// TwinCAT 3 PLC project PLC
// ProgramVersion: 3.1.4024.0
// libraries:
//   SPT Base Types, * (Beckhoff Automation LLC)
//   SPT Components, * (Beckhoff Automation LLC)
//   SPT Diagnostic, * (Beckhoff Automation LLC)
//   SPT EtherCat, * (Beckhoff Automation LLC)
//   SPT Event Logger, * (Beckhoff Automation LLC)
//   SPT Kinematics, * (Beckhoff Automation LLC)
//   SPT Motion Control, * (Beckhoff Automation LLC)
//   SPT NCI, * (Beckhoff Automation LLC)
//   SPT Utilities, * (Beckhoff Automation LLC)
//   SPT Vision, * (Beckhoff Automation LLC)
//   SPT XTS, * (Beckhoff Automation LLC)
//   Tc2_Standard, * (Beckhoff Automation GmbH)
//   Tc2_System, * (Beckhoff Automation GmbH)
//   Tc3_EventLogger, * (Beckhoff Automation GmbH)
//   Tc3_Module, * (Beckhoff Automation GmbH)
//   Tc3_PackML_V2, * (Beckhoff Automation GmbH)
// project tree:
//   / GlobalTextList.TcGTLO (not stored), PlcTask.TcTTO (not stored), Visualization Manager.TcVMO (not stored)
//   Machine/01_MachineModule/ Machine.TcPOU
//   Machine/02_EquipmentModules/ InfeedModule.TcPOU, OutfeedModule.TcPOU, ProcessModule.TcPOU
//   Machine/03_Components/ SampleComponent.TcPOU
//   POUs/ MAIN.TcPOU
//   VISUs/ Visualization.TcVIS
// real-time tasks:
//   TASK PlcTask: cycle T#10ms, priority 20, ADS port 350

// ---- Machine/01_MachineModule/Machine.TcPOU
FUNCTION_BLOCK Machine EXTENDS FB_PackML_BaseModule
VAR
	//EMs
	Infeed	: InfeedModule	:= (Name := 'Infeed');
	Process : ProcessModule := (Name := 'Process');
	Outfeed : OutfeedModule := (Name := 'Outfeed');

	//
	_StopRequestFromEM : BOOL;
END_VAR

//! @summary This method serves as the entry point for all underlying FB logic

//! @description This method should be called cyclically by descendant function blocks by invoking <c>SUPER^.CyclicLogic()</c>.  Alternatively, the contents of this method could be reimplemented entirely in which case a call to this method would not be necessary.
METHOD PUBLIC CyclicLogic
VAR
	i : UDINT;
END_VAR
IF NOT _InitComplete THEN
	_InitComplete := Initialize();
	RETURN;
END_IF

//Decide when to Stop Machine based on EM Stop Request
IF _StopRequestFromEM AND Outfeed.CurrentState = E_PMLState.ePMLState_Complete THEN
	ChangeState(State := E_PMLCommand.ePMLCommand_Abort);
	Process.StopRequestToMM := FALSE;
END_IF

//
SUPER^.CyclicLogic();
END_METHOD

// Automatically enables and disables HMI control based on the PackML mode
METHOD PROTECTED HMIPermissions

// This method is called cyclically by CyclicLogic()
AllowHMIControl(ThisModuleOnly := TRUE);
END_METHOD

//! @summary Basic module initialization logic
METHOD PROTECTED Initialize : BOOL;
VAR
	i						 : UDINT;
	varInfo					 : __SYSTEM.VAR_INFO;
	AllSubUnitsInitialized	 : BOOL := TRUE;
	AllComponentsInitialized : BOOL := TRUE;
END_VAR

//! @description This method is called by <c>CyclicLogic()</c> as required
Initialize := FALSE;
CASE DescendantSequenceState OF
	0: //Register Modules
		RegisterSubmodule(Infeed);
		RegisterSubmodule(Process);
		RegisterSubmodule(Outfeed);

		//Register Components

		//Setup Config
		_LogModeChanges			:= FALSE;
		_LogStateChanges		:= FALSE;
		DescendantSequenceState := DescendantSequenceState + 10;

	10: // Copy Mode names
		FOR i := 1 TO 10 DO
			ModeNames[i] := F_UnitModeToString(UDINT_TO_DINT(i));
		END_FOR

		DescendantSequenceState := DescendantSequenceState + 10;

	20: // Call the Super 
		IF SUPER^.Initialize() THEN
			Initialize := TRUE;
		END_IF
END_CASE
END_METHOD

//! @summary This method monitors <b>submodules</b> within this PackML module and initiates fault responses as required
METHOD PROTECTED SubModuleMonitor : BOOL
VAR
	AlarmResponses : ARRAY[0..4] OF E_AlarmResponse; //Temporary response array	
	i			   : UDINT;
END_VAR

//! @description This method is called cyclically by <c>CyclicLogic()</c>
IF Process.StopRequestToMM THEN
	_StopRequestFromEM := TRUE;
ELSE
	_StopRequestFromEM := FALSE;
END_IF

SUPER^.SubModuleMonitor();
END_METHOD

END_FUNCTION_BLOCK

// ---- Machine/02_EquipmentModules/InfeedModule.TcPOU
FUNCTION_BLOCK InfeedModule EXTENDS FB_PackML_BaseModule
VAR
END_VAR

//! @summary This method serves as the entry point for all underlying FB logic

//! @description This method should be called cyclically by descendant function blocks by invoking <c>SUPER^.CyclicLogic()</c>.  Alternatively, the contents of this method could be reimplemented entirely in which case a call to this method would not be necessary.
METHOD PUBLIC CyclicLogic
VAR
	i : UDINT;
END_VAR
IF NOT _InitComplete THEN
	_InitComplete := Initialize();
	RETURN;
END_IF

SUPER^.CyclicLogic();
END_METHOD

//! @summary Basic module initialization logic
METHOD PROTECTED Initialize : BOOL;
VAR
	i						 : UDINT;
	varInfo					 : __SYSTEM.VAR_INFO;
	AllSubUnitsInitialized	 : BOOL := TRUE;
	AllComponentsInitialized : BOOL := TRUE;
END_VAR

//! @description This method is called by <c>CyclicLogic()</c> as required
Initialize := FALSE;
CASE DescendantSequenceState OF
	0: //Register Modules

		//Register Components

		//Setup Config
		_LogModeChanges			:= FALSE;
		_LogStateChanges		:= FALSE;
		DescendantSequenceState := DescendantSequenceState + 10;

	10: // Copy Mode names
		FOR i := 1 TO 10 DO
			ModeNames[i] := F_UnitModeToString(UDINT_TO_DINT(i));
		END_FOR

		DescendantSequenceState := DescendantSequenceState + 10;

	20: // Call the Super 
		IF SUPER^.Initialize() THEN
			Initialize := TRUE;
		END_IF
END_CASE
END_METHOD

END_FUNCTION_BLOCK

// ---- Machine/02_EquipmentModules/ProcessModule.TcPOU
FUNCTION_BLOCK ProcessModule EXTENDS FB_PackML_BaseModule
VAR
	Component : SampleComponent := (Name := 'Sample Component');

	//
	_StopRequestToMM : BOOL;
END_VAR

//! @summary This method serves as the entry point for all underlying FB logic

//! @description This method should be called cyclically by descendant function blocks by invoking <c>SUPER^.CyclicLogic()</c>.  Alternatively, the contents of this method could be reimplemented entirely in which case a call to this method would not be necessary.
METHOD PUBLIC CyclicLogic
VAR
	i : UDINT;
END_VAR
IF NOT _InitComplete THEN
	_InitComplete := Initialize();
	RETURN;
END_IF

SUPER^.CyclicLogic();
END_METHOD

//! @summary Basic module initialization logic
METHOD PROTECTED Initialize : BOOL;
VAR
	i						 : UDINT;
	varInfo					 : __SYSTEM.VAR_INFO;
	AllSubUnitsInitialized	 : BOOL := TRUE;
	AllComponentsInitialized : BOOL := TRUE;
END_VAR

//! @description This method is called by <c>CyclicLogic()</c> as required
Initialize := FALSE;
CASE DescendantSequenceState OF
	0: //Register Modules

		//Register Components
		RegisterComponent(Component);

		//Setup Config
		_LogModeChanges			:= FALSE;
		_LogStateChanges		:= FALSE;
		DescendantSequenceState := DescendantSequenceState + 10;

	10: // Copy Mode names
		FOR i := 1 TO 10 DO
			ModeNames[i] := F_UnitModeToString(UDINT_TO_DINT(i));
		END_FOR

		DescendantSequenceState := DescendantSequenceState + 10;

	20: // Call the Super 
		IF SUPER^.Initialize() THEN
			Initialize := TRUE;
		END_IF
END_CASE
END_METHOD

//! @summary Provides fault reaction logic where the module state is driven to the <b>Stopping</b> state at the next available opportunity
METHOD PROTECTED StopControlled

(*! <description> No error is thrown by this fault reaction.
	<b> TODO: Needs implementation </b> </description>*)

//! @description This method is called by <c>ComponentMonitor()</c> or <c>SubModuleMonitor()</c> as required
//Add code here for Controlled Stop, this code will not impact the other EMs

//Add code here to notify the MM that the Module is stopping and the Machine should stop also (* this is optional *)
_StopRequestToMM := TRUE;

//
SUPER^.StopControlled();
END_METHOD

PROPERTY StopRequestToMM : BOOL
GET
StopRequestToMM := _StopRequestToMM;
END_GET
SET
_StopRequestToMM := StopRequestToMM;
END_SET
END_PROPERTY

END_FUNCTION_BLOCK

// ---- Machine/03_Components/SampleComponent.TcPOU
FUNCTION_BLOCK SampleComponent EXTENDS FB_ComponentBase
VAR
	//Alarms
	ComponentAlarms : ARRAY[1..ALARM_COUNT] OF FB_TcAlarm;
	testError		: BOOL;
END_VAR

VAR CONSTANT
	ALARM_COUNT : INT := 6;
END_VAR

//! @summary Initializes event function blocks using this components's name
METHOD PROTECTED CreateEvents

//! @description This method is called by <c>Initialize()</c> as required
F_CreateAllEventsInClass(Alarms		:= ComponentAlarms,
						 ClassSize	:= SIZEOF(TC_Events.ComponentEvents),
						 pInitEvent := ADR(TC_EVENTS.ComponentEvents.InitReferenceEvent),
						 Prefix		:= Name);

SUPER^.CreateEvents();
END_METHOD

//! @summary This method serves as the entry point for all underlying FB logic
METHOD PUBLIC CyclicLogic

//! @description This method should be called cyclically by descendant function blocks by invoking <c>SUPER^.CyclicLogic()</c>.  Alternatively, the contents of this method could be reimplemented entirely in which case a call to this method would not be necessary.
IF NOT _InitComplete THEN
	_InitComplete := Initialize();
	RETURN;
END_IF

SUPER^.CyclicLogic();

(*
*
*		Code must be after SUPER^.CyclicLogic();
*
*)

(* Update alarm severity from this component *)
_CurrentAlarmSeverity := F_GetMaxSeverityRaised(Alarms := ComponentAlarms, CurrentSeverity := _CurrentAlarmSeverity);
_Error				  := _CurrentAlarmSeverity >= TcEventSeverity.Error;
END_METHOD

//! @summary Basic component initialization logic
METHOD PROTECTED Initialize : BOOL;

//! @description This method is called by <c>CyclicLogic()</c> as required
//Setting the Fault Response Definition here will cause the EM that uses this Component to call the StopControlled method of the EM
_ParentFaultResponseDefinitions[TcEventSeverity.Error] := E_AlarmResponse.Stop_Controlled;

//
Initialize := SUPER^.Initialize();
END_METHOD

//! Provides basic error detection and event handling for this component
METHOD PROTECTED Monitoring
(*! @descriptionThis method is called cyclically by <c>CyclicLogic()</c>*)
VAR
	i : INT;
END_VAR
IF testError AND NOT ComponentAlarms[5].bRaised THEN
	RaiseAlarm2Args(ComponentAlarms[5], CONCAT('Error ID: ', TO_STRING(_ErrorID)), '');
END_IF

SUPER^.Monitoring();
END_METHOD

METHOD RaiseAlarm2Args
VAR_IN_OUT
	Alarm : FB_TcAlarm; //Alarm to be raised
END_VAR

VAR_INPUT
	String_1 : STRING; //First String Parameter (The Name of this component will be applied first automatically)
	String_2 : STRING; //Second String Parameter
END_VAR
F_RaiseAlarmWithStringParameters(Alarm	  := Alarm,
								 String_1 := Name,
								 String_2 := String_1,
								 String_3 := String_2);
END_METHOD

//! @summary Clears error flags and error IDs for this component

//Typically called by the EMs SUPER^.Clearing Method
METHOD PUBLIC Reset : BOOL
F_ClearAllEventsInClass(Alarms := ComponentAlarms);
IF SUPER^.Reset() THEN
	_Error	 := FALSE;
	_ErrorID := 0;
	Reset	 := TRUE;
END_IF
END_METHOD

END_FUNCTION_BLOCK

// ---- Machine/02_EquipmentModules/OutfeedModule.TcPOU
FUNCTION_BLOCK OutfeedModule EXTENDS FB_PackML_BaseModule
VAR
	testComplete : BOOL;
END_VAR

//! @summary This method serves as the entry point for all underlying FB logic

//! @description This method should be called cyclically by descendant function blocks by invoking <c>SUPER^.CyclicLogic()</c>.  Alternatively, the contents of this method could be reimplemented entirely in which case a call to this method would not be necessary.
METHOD PUBLIC CyclicLogic
VAR
	i : UDINT;
END_VAR
IF NOT _InitComplete THEN
	_InitComplete := Initialize();
	RETURN;
END_IF

SUPER^.CyclicLogic();

//
IF testComplete THEN
	testComplete := FALSE;
	Trace('Outfeed changing state to Complete');
	ChangeState(State := E_PMLCommand.ePMLCommand_Complete);
END_IF
END_METHOD

//! @summary Basic module initialization logic
METHOD PROTECTED Initialize : BOOL;
VAR
	i						 : UDINT;
	varInfo					 : __SYSTEM.VAR_INFO;
	AllSubUnitsInitialized	 : BOOL := TRUE;
	AllComponentsInitialized : BOOL := TRUE;
END_VAR

//! @description This method is called by <c>CyclicLogic()</c> as required
Initialize := FALSE;
CASE DescendantSequenceState OF
	0: //Register Modules

		//Register Components

		//Setup Config
		_LogModeChanges			:= FALSE;
		_LogStateChanges		:= FALSE;
		DescendantSequenceState := DescendantSequenceState + 10;

	10: // Copy Mode names
		FOR i := 1 TO 10 DO
			ModeNames[i] := F_UnitModeToString(UDINT_TO_DINT(i));
		END_FOR

		DescendantSequenceState := DescendantSequenceState + 10;

	20: // Call the Super 
		IF SUPER^.Initialize() THEN
			Initialize := TRUE;
		END_IF
END_CASE
END_METHOD

END_FUNCTION_BLOCK

// ---- POUs/MAIN.TcPOU
PROGRAM MAIN
VAR
	Machine : Machine := (Name := 'Machine');
END_VAR

// All sample code provided by Beckhoff Automation LLC are for illustrative purposes only and are provided “as is” and without any warranties, express or implied. Actual implementations in applications will vary significantly. Beckhoff Automation LLC shall have no liability for, and does not waive any rights in relation to, any code samples that it provides or the use of such code samples for any purpose.

(*

This code is intended to be a simple example of how to perform a controlled stop of a machine when one EM has an error.
The idea is that the EM with an Errored Component will call its StopControlled method and set a flag that is read by the MM, signaling that the machine needs to stop.
Once the required EMs have completed (CurrentState = Completed), the machine can then issue an abort command.



//These are the possible alarm responses, each of these has a corresponding method that will be called from the SubModuleMonitor() or ComponentMonitor()

TYPE E_AlarmResponse : (
		Abort_ImmediateError,
		Abort_Immediate,
		Stop_Immediate,
		Stop_Controlled,
		Hold_Immediate,
		Hold_Controlled,
		Suspend_Immediate,
		Suspend_Controlled,
		NoResponse - No corresponding Method
	);
END_TYPE


//Each Fault in the type system has a severity level
TcEventSeverity.Verbose
TcEventSeverity.Info
TcEventSeverity.Warning
TcEventSeverity.Error
TcEventSeverity.Critical

//The array indexes below 0..4 correspond to the above severity levels
//These are the defaults, therefore Verbose, Info, and Warning have NoResponse
	while Error and Critical are set to AbortImmediateError
	
_ParentFaultResponseDefinitions : ARRAY[0..4] OF E_AlarmResponse := 
	[E_AlarmResponse.NoResponse, 
	E_AlarmResponse.NoResponse, 
	E_AlarmResponse.NoResponse, 
	E_AlarmResponse.Abort_ImmediateError, 
	E_AlarmResponse.Abort_ImmediateError];

In order to have a component set to StopControlled, change the _ParentFaultResponseDefinitions in the Initialize method of that component
_ParentFaultResponseDefinitions[TcEventSeverity.Error] := E_AlarmResponse.Stop_Controlled;

//The StopControlled method of the base class must then be overridden.
Include any code needed to handle the other components within the EM and then call the SUPER^.StopControlled()
This will place the EM into State = Stopped

In order to stop the entire machine after each EM has processed its current product a flag is set in the EM, StopRequestToMM.
This flag is monitored by the SubModuleMonitor method of the MM, if TRUE it sets a local variable _StopRequestFromEM

IF Process.StopRequestToMM THEN
	_StopRequestFromEM := TRUE;
END_IF


In the CyclicLogic method of the MM, if the StopRequest is TRUE and the required EMs are in State = Complete
the MM will issue an abort command to itself, which by default will cause all EMs to abort

IF _StopRequestFromEM AND Outfeed.CurrentState = E_PMLState.ePMLState_Complete THEN
	ChangeState(State := E_PMLCommand.ePMLCommand_Abort);
END_IF
	


Code to take note of:
SampleComponent.Initialize()
ProcessModule.StopControlled()
ProcessModule.StopRequestToMM.Get
Machine.SubModuleMonitor()
Machine.CyclicLogic()


To run the test:
1. Toggle resetStateMachine in MAIN - this will place the MM and all EMs in Production-Execute
2. Verify that all EMs are in Production-Execute
3. Toggle testError in SampleComponent.Monitoring()
4. Verify that the Process Module is in Stopped, and note that the other EMs are still in Production-Execute
5. Toggle testComplete in OutfeedModule.CyclicLogic()
6. Verify that the MM and all EMs are in Production-Aborted
7. Toggle testError in SampleComponent.Monitoring() - failure to turn off the error will cause the state machine of the ProcessModule to get stuck, you can use the abort command to recover from this situation
8. Return to step 1

*)

//This is for debug only and should be removed
_AppInfo.KeepOutputsOnBP := TRUE;

//
Machine.CyclicLogic();

END_PROGRAM

// ---- VISUs/Visualization.TcVIS
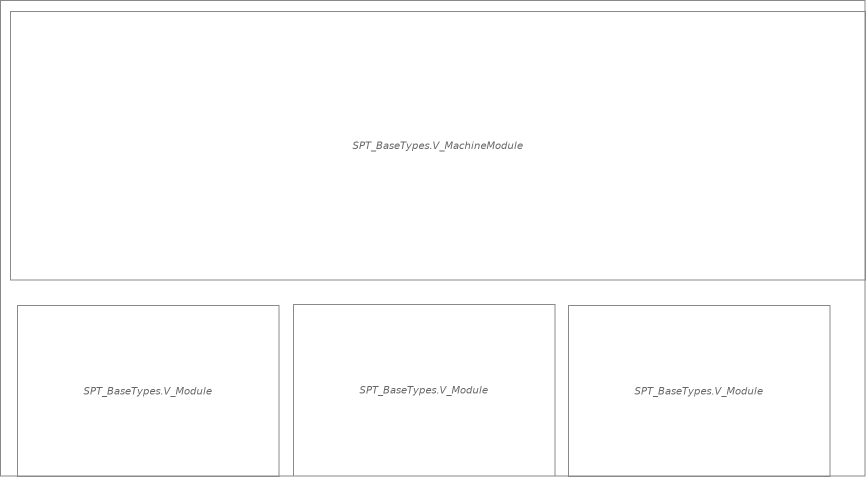
VISUALIZATION Visualization  // 866x477
    Frame (10,11 856x269)
        shows SPT_BaseTypes.V_MachineModule(HMI := MAIN.Machine.PackMLBaseModule_HMI)
    Frame (17,305 262x172)
        shows SPT_BaseTypes.V_Module(HMI := MAIN.Machine.Infeed.PackMLBaseModule_HMI)
    Frame (293,304 262x172)
        shows SPT_BaseTypes.V_Module(HMI := MAIN.Machine.Process.PackMLBaseModule_HMI)
    Frame (568,305 262x172)
        shows SPT_BaseTypes.V_Module(HMI := MAIN.Machine.Outfeed.PackMLBaseModule_HMI)
END_VISUALIZATION
